TYPE ST_TU_DataEmulation :
(**************************************************************************************
 * 	Application		:	BoxControl Framework
 *	Revision		:	$Revision: 412414 $
 *	Revision date	:	$Date: 2018-08-17 07:57:24 +0200 (Fr., 17 Aug 2018) $
 *	Last changed by	:	$Author: d7herza $
 *	URL				:	$URL: http://almscdc.swisslog.com/repo/SWPD/Development/BoxControlFramework/20_Release/trunk/01_Software/BCF/BCF/JumpStart/20_Product/11_Emu/10_Base/10_Lib/10_Conv/01_DUTs/ST_TU_DataEmulation.TcDUT $
 *
 *	Purpose			:	TU Data
 *
 * ------------------------------------------------------------------------------------
 *	Copyright Swisslog [IP AG], Switzerland. All rights reserved.
 * 
 * ------------------------------------------------------------------------------------
 *	
 * 	Revision History: 
 *
 * 	VERSION			DATE			INITIALS			DESCRIPTION
 *	0.1				01.01.2001		swl					Example
 *
 **************************************************************************************)
STRUCT
	DataSet			: ST_DataSetEmulation; // DataSet
	Label			: ST_LabelEmulation; // Label
	TimeStamp		: ST_TimeStamp; // TimeStamp 
END_STRUCT
END_TYPE

(* stored: Version 1.1.0.1, ProductVersion 3.1.4022.12
   DUT ST_TU_DataEmulation: Id {264e4b91-f97b-4e53-81d0-f59cc18bca76} *)
